Universal Robots PolyScope program: beksflaeks.urp

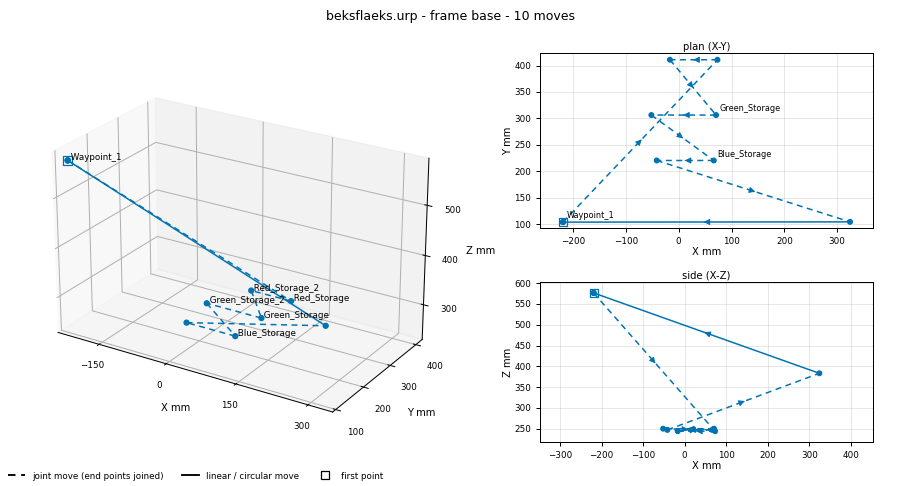
[picture p0: tool path of beksflaeks.urp in frame base, 10 of 11 moves have a stored position in this frame; points joined in program order, loops and branches not executed]
Program beksflaeks (installation=default directory=/programs/usbdisk_1/new createdIn=3.9.1.64192 lastSavedIn=3.9.1.64192 robotSerialNumber=2016331617)
Calibrated DH parameters: a=[-0.000045, -0.22956, -0.153032, 0.000019, 0.0001, 0]; d=[0.152163, -856.35044, 904.692211, -48.229373, 0.085425, 0.082565]; alpha=[1.571202, -0.000097, 0.003084, 1.571016, -1.571253, 0]; deltaTheta=[-0.00003, 0.346154, 0.426056, -0.772366, 0.00006, 0.000029]
BeforeStart
  Loop Forever
    Script: conres = socket_open("192.168.137.1",23)
    Script: textmsg(conres)
    If conres ≟  True
      Script: break
  Script: targetPos=p[0, 0, 0, 0, 0, 0]
  Script: receiveFromServ=[0, 0, 0, 0, 0, 0, 0, 0]
Robot Program (runOnlyOnce=false)
  Set DigitalOutput pin=tool_out[0]; digitalValue=0
  MoveJ speed 60 deg/s, acceleration 80 deg/s^2 (useActiveTCP=true)
    Waypoint Waypoint_1: TCP in base x=-218.947 y=103.634 z=576.492 mm, rx=-0.8555 ry=-1.2749 rz=-0.1412 rad; joints [-62.287, -105.827, 77.47, -154.059, -66.74, -60.096] deg
  Script: sendToServer="Klar"
  Script: socket_send_string(sendToServer)
  Loop While (checkContinuously=false) expression=conres≟ True
    Script: receiveFromServ=socket_read_ascii_float(7)
    Script: textmsg(receiveFromServ)
    If receiveFromServ[7]≟1
      Script: break
    ElseIf receiveFromServ[7]≟2
      Script: break
    ElseIf receiveFromServ[7]≟3
      Script: break
    ElseIf receiveFromServ[7]≟4
      Script: break
  Loop Forever
    Script: targetPos=p[receiveFromServ[1],receiveFromServ[2],receiveFromServ[3],receiveFromServ[4],receiveFromServ[5],receiveFromServ[6]]
    Script: textmsg(targetPos)
    If targetPos≠p[0, 0, 0, 0, 0, 0]
      MoveL speed 250 mm/s, acceleration 1200 mm/s^2 (useActiveTCP=true) feature=Base
        Waypoint Waypoint (Variable): variable=targetPos
      Script: break
  Set ExpressionOutput pin=tool_out[0]; expression=True
  Wait Sleep waitTime=2
  MoveJ speed 60 deg/s, acceleration 80 deg/s^2 (useActiveTCP=true)
    Waypoint Waypoint_1: TCP in base x=-218.947 y=103.634 z=576.492 mm, rx=-0.8555 ry=-1.2749 rz=-0.1412 rad; joints [-62.287, -105.827, 77.47, -154.059, -66.74, -60.096] deg
  Wait Sleep waitTime=2
  If receiveFromServ[7]≟1
    If Red≟0
      MoveJ speed 60 deg/s, acceleration 80 deg/s^2 (useActiveTCP=true)
        Waypoint Red_Storage: TCP in base x=73.399 y=410.879 z=243.753 mm, rx=-2.6828 ry=-1.565 rz=0.0637 rad; joints [-116.419, -63.852, 75.621, -100.933, -86.913, -86.822] deg
        Set ExpressionOutput pin=tool_out[0]; expression=False
        Wait Sleep waitTime=1
        Set IncrementVariable installationVariable=Red
    ElseIf Red≠0
      MoveJ speed 60 deg/s, acceleration 80 deg/s^2 (useActiveTCP=true)
        Waypoint Red_Storage_2: TCP in base x=-16.551 y=410.893 z=243.78 mm, rx=-2.6827 ry=-1.5649 rz=0.0635 rad; joints [-104.259, -65.548, 78.427, -102.698, -86.806, -74.639] deg
        Set ExpressionOutput pin=tool_out[0]; expression=False
        Wait Sleep waitTime=1
  ElseIf receiveFromServ[7]≟2
    If Green≟0
      MoveJ speed 60 deg/s, acceleration 80 deg/s^2 (useActiveTCP=true)
        Waypoint Green_Storage: TCP in base x=70.718 y=306.264 z=249.848 mm, rx=-2.7016 ry=-1.4787 rz=0.0435 rad; joints [-125.132, -89.524, 106.948, -107.552, -86.025, -92.369] deg
        Set ExpressionOutput pin=tool_out[0]; expression=False
        Wait Sleep waitTime=1
        Set IncrementVariable installationVariable=Green
    ElseIf Green≠0
      MoveJ speed 60 deg/s, acceleration 80 deg/s^2 (useActiveTCP=true)
        Waypoint Green_Storage_2: TCP in base x=-51.686 y=306.259 z=249.829 mm, rx=-2.7018 ry=-1.4787 rz=0.0435 rad; joints [-102.735, -90.747, 108.788, -109.634, -86.367, -69.922] deg
        Set ExpressionOutput pin=tool_out[0]; expression=False
        Wait Sleep waitTime=1
  ElseIf receiveFromServ[7]≟3
    If Blue≟0
      MoveJ speed 60 deg/s, acceleration 80 deg/s^2 (useActiveTCP=true)
        Waypoint Blue_Storage: TCP in base x=66.478 y=220.285 z=246.895 mm, rx=-2.7077 ry=-1.5077 rz=0.0571 rad; joints [-137.325, -112.52, 124.913, -100.928, -87.046, -105.446] deg
        Set ExpressionOutput pin=tool_out[0]; expression=False
        Wait Sleep waitTime=1
        Set IncrementVariable installationVariable=Blue
    ElseIf Blue≠0
      MoveJ speed 60 deg/s, acceleration 80 deg/s^2 (useActiveTCP=true)
        Waypoint Blue_Storage_2: TCP in base x=-41.487 y=220.272 z=246.895 mm, rx=-2.7076 ry=-1.5078 rz=0.0571 rad; joints [-110.926, -115.037, 126.823, -101.738, -86.682, -79.016] deg
        Set ExpressionOutput pin=tool_out[0]; expression=False
        Wait Sleep waitTime=1
  ElseIf receiveFromServ[7]≟4
    MoveJ speed 60 deg/s, acceleration 80 deg/s^2 (useActiveTCP=true)
      Waypoint Skrald: TCP in base x=324.295 y=104.113 z=383.107 mm, rx=-2.9845 ry=-0.398 rz=-0.2817 rad; joints [-183.781, -86.97, 72.213, -84.486, -81.166, -108.163] deg
      Set ExpressionOutput pin=tool_out[0]; expression=False
      Wait Sleep waitTime=1
  Wait Sleep waitTime=1
  Script: targetPos=p[0, 0, 0, 0, 0, 0]
  MoveL speed 250 mm/s, acceleration 1200 mm/s^2 (useActiveTCP=true) feature=Base
    Waypoint Waypoint_1: TCP in base x=-218.947 y=103.634 z=576.492 mm, rx=-0.8555 ry=-1.2749 rz=-0.1412 rad; joints [-62.287, -105.827, 77.47, -154.059, -66.74, -60.096] deg
